// TwinCAT 3 PLC project HXR_GATT
// ProgramVersion: 3.1.4022.4
// libraries:
//   L2SI Vacuum Library, * (SLAC)
//   LCLS General, * (SLAC)
//   Tc2_ControllerToolbox, * (Beckhoff Automation GmbH)
//   Tc2_DataExchange, * (Beckhoff Automation GmbH)
//   Tc2_EtherCAT, * (Beckhoff Automation GmbH)
//   Tc2_Standard, * (Beckhoff Automation GmbH)
//   Tc2_System, * (Beckhoff Automation GmbH)
//   Tc2_Utilities, * (Beckhoff Automation GmbH)
//   Tc3_Module, * (Beckhoff Automation GmbH)
// project tree:
//   DUTs/ E_PositionState.TcDUT (not stored), ST_MPA.TcDUT, ST_PressureSensor.TcDUT
//   GVLs/ GVL_Devices.TcGVL, GVL_ILK.TcGVL, GVL_Sensors.TcGVL (not stored)
//   / PlcTask.TcTTO
//   POUs/ DIAGNOSTICS.TcPOU (not stored), FB_MPA.TcPOU, FB_PressureSensor_PX219.TcPOU (not stored), MAIN.TcPOU, PRG_ACTUATORS.TcPOU, PRG_DIFF_PUMP.TcPOU, PRG_GATT.TcPOU, PRG_GEM.TcPOU, PRG_GEM1.TcPOU, PRG_ILK.TcPOU, PRG_PMPS.TcPOU, PRG_ROOTS.TcPOU, PRG_SENSORS.TcPOU (not stored)
// real-time tasks:
//   TASK PlcTask: cycle T#10ms, priority 20, ADS port 350
// I/O:
//   DEVICE AT1L0 (EtherCAT), AmsNetId 134.79.72.124.4.1
//     PLC_AT1L0 (EK1200) [EK1200-5000 EtherCAT Power supply (2A E-Bus)]
//       PLC_EL_1 (EL2088) [EL2088 8Ch. Dig. Output 24V, 0.5A, switching to negative]
//       PLC_EL_2 (EL1088) [EL1088 8Ch. Dig. Input 24V, 3ms, negative]
//       PLC_EL_3 (EL1088) [EL1088 8Ch. Dig. Input 24V, 3ms, negative]
//       PLC_EL_4 (EL2088) [EL2088 8Ch. Dig. Output 24V, 0.5A, switching to negative]
//       PLC_EL_5 (EL1088) [EL1088 8Ch. Dig. Input 24V, 3ms, negative]
//       PLC_EL_6 (EL1088) [EL1088 8Ch. Dig. Input 24V, 3ms, negative]
//       PLC_EL_7 (EL9187) [EL9187 Potential Connection, 8 x Ground]
//       PLC_EL_8 (EL2088) [EL2088 8Ch. Dig. Output 24V, 0.5A, switching to negative]
//       PLC_EL_9 (EL1088) [EL1088 8Ch. Dig. Input 24V, 3ms, negative]
//       PLC_EL_10 (EL1088) [EL1088 8Ch. Dig. Input 24V, 3ms, negative]
//       PLC_EL_11 (EL2088) [EL2088 8Ch. Dig. Output 24V, 0.5A, switching to negative]
//       PLC_EL_12 (EL1088) [EL1088 8Ch. Dig. Input 24V, 3ms, negative]
//       PLC_EL_13 (EL1088) [EL1088 8Ch. Dig. Input 24V, 3ms, negative]
//       PLC_EL_14 (EL9187) [EL9187 Potential Connection, 8 x Ground]
//       PLC_EL_15 (EL2624) [EL2624 4Ch. Relay Output, NO (125V AC / 30V DC)]
//       PLC_EL_16 (EL2202) [EL2202 2Ch. Dig. Output 24V, 0.5A]
//       PLC_EL_17 (EL6692) [EL6692 EtherCAT Bridge terminal (Primary)]
//       PLC_EK_18 (EK1110) [EK1110 EtherCAT extension]
//     DRL_MKS (EK1100) [EK1100 EtherCAT Coupler (2A E-Bus)]
//       MKS_E1 (EL3064) [EL3064 4Ch. Ana. Input 0-10V]
//       MKS_E2 (EL3064) [EL3064 4Ch. Ana. Input 0-10V]
//       MKS_E3 (EL2794) [EL2794 4Ch. Dig. Output 24V AC/DC, 2A, short-circuit-proof]
//       MKS_E4 (EL3064) [EL3064 4Ch. Ana. Input 0-10V]
//       MKS_E5 (EL3064) [EL3064 4Ch. Ana. Input 0-10V]
//       MKS_E6 (EL2794) [EL2794 4Ch. Dig. Output 24V AC/DC, 2A, short-circuit-proof]
//       MKS_E7 (EL3064) [EL3064 4Ch. Ana. Input 0-10V]
//       MKS_E8 (EL3064) [EL3064 4Ch. Ana. Input 0-10V]
//       MKS_E9 (EL2794) [EL2794 4Ch. Dig. Output 24V AC/DC, 2A, short-circuit-proof]
//       MKS_E10 (EL3064) [EL3064 4Ch. Ana. Input 0-10V]
//       MKS_E11 (EL3064) [EL3064 4Ch. Ana. Input 0-10V]
//       MKS_E12 (EL2794) [EL2794 4Ch. Dig. Output 24V AC/DC, 2A, short-circuit-proof]
//       MKS_E13 (EL3064) [EL3064 4Ch. Ana. Input 0-10V]
//       MKS_E14 (EL3064) [EL3064 4Ch. Ana. Input 0-10V]
//       MKS_E15 (EL2794) [EL2794 4Ch. Dig. Output 24V AC/DC, 2A, short-circuit-proof]
//     L0S3_PNL_01_EB_1 (EP2338-0002) [EP2338-0002 8 Ch. Dig. Input/Output 24V, 0,5A, M12]
//     L0S3_PNL_01_EB_2 (EP2338-0002) [EP2338-0002 8 Ch. Dig. Input/Output 24V, 0,5A, M12]
//     L0S3_PNL_01_EB_3 (EP2338-0002) [EP2338-0002 8 Ch. Dig. Input/Output 24V, 0,5A, M12]
//     L0S3_PNL_01_EB_4 (EP2338-0002) [EP2338-0002 8 Ch. Dig. Input/Output 24V, 0,5A, M12]
//     L0S3_PNL_01_EB_5 (EP3174-0002) [EP3174-0002 4Ch. Ana. Input +/-10V, 0-10V, 0/4-20mA configurable]
//     L0S3_PNL_01_EB_6 (EP3174-0002) [EP3174-0002 4Ch. Ana. Input +/-10V, 0-10V, 0/4-20mA configurable]
//     L0S3_PNL_02_EB_1 (EP2338-0002) [EP2338-0002 8 Ch. Dig. Input/Output 24V, 0,5A, M12]
//     L0S3_PNL_02_EB_2 (EP2338-0002) [EP2338-0002 8 Ch. Dig. Input/Output 24V, 0,5A, M12]
//     L0S3_PNL_02_EB_3 (EP4374-0002) [EP4374-0002 2Ch. Ana. Input +/-10V, 0-10V, 0/4-20mA configurable; 2Ch. Ana. Output +/-10V, 0-10V, 0/4-20mA configurable]
//     L0S3_PNL_02_EB_4 (EP3174-0002) [EP3174-0002 4Ch. Ana. Input +/-10V, 0-10V, 0/4-20mA configurable]
//     L0S3_PNL_02_EB_5 (EP2624-0002) [EP2624-0002 4Ch. Relay Output, NO (125V AC / 30V DC)]
//     L0S3_PNL_03_EB_1 (EP2338-0002) [EP2338-0002 8 Ch. Dig. Input/Output 24V, 0,5A, M12]
//     L0S3_PNL_03_EB_2 (EP2338-0002) [EP2338-0002 8 Ch. Dig. Input/Output 24V, 0,5A, M12]
//     L0S3_PNL_03_EB_3 (EP2338-0002) [EP2338-0002 8 Ch. Dig. Input/Output 24V, 0,5A, M12]
//     L0S3_PNL_03_EB_4 (EP3174-0002) [EP3174-0002 4Ch. Ana. Input +/-10V, 0-10V, 0/4-20mA configurable]
//     L0S3_PNL_03_EB_5 (EP3174-0002) [EP3174-0002 4Ch. Ana. Input +/-10V, 0-10V, 0/4-20mA configurable]
//     L0S3_PNL_03_EB_6 (EP2624-0002) [EP2624-0002 4Ch. Relay Output, NO (125V AC / 30V DC)]
//     L0S3_PNL_03_EB_7 (EP2338-0002) [EP2338-0002 8 Ch. Dig. Input/Output 24V, 0,5A, M12]
//     L0S3_PNL_03_EB_8 (EP2624-0002) [EP2624-0002 4Ch. Relay Output, NO (125V AC / 30V DC)]
//     L0S3_PNL_03_EB_9 (EP2338-0002) [EP2338-0002 8 Ch. Dig. Input/Output 24V, 0,5A, M12]
//     L0S6_PNL_04_EB_1 (EP2338-0002) [EP2338-0002 8 Ch. Dig. Input/Output 24V, 0,5A, M12]
//     L0S6_PNL_04_EB_2 (EP3174-0002) [EP3174-0002 4Ch. Ana. Input +/-10V, 0-10V, 0/4-20mA configurable]
//     L0S6_PNL_04_EB_3 (EP4374-0002) [EP4374-0002 2Ch. Ana. Input +/-10V, 0-10V, 0/4-20mA configurable; 2Ch. Ana. Output +/-10V, 0-10V, 0/4-20mA configurable]
//     L0S6_PNL_04_EB_4 (EP2338-0002) [EP2338-0002 8 Ch. Dig. Input/Output 24V, 0,5A, M12]
//     L0S6_PNL_04_EB_5 (EP2338-0002) [EP2338-0002 8 Ch. Dig. Input/Output 24V, 0,5A, M12]
//     L0S6_PNL_04_EB_6 (EP2338-0002) [EP2338-0002 8 Ch. Dig. Input/Output 24V, 0,5A, M12]
//     L0S6_PNL_04_EB_7 (EP2338-0002) [EP2338-0002 8 Ch. Dig. Input/Output 24V, 0,5A, M12]
//     L0S6_PNL_04_EB_8 (EP2338-0002) [EP2338-0002 8 Ch. Dig. Input/Output 24V, 0,5A, M12]
//     L0S6_PNL_01_EB_1 (EP2338-0002) [EP2338-0002 8 Ch. Dig. Input/Output 24V, 0,5A, M12]
//     L0S6_PNL_01_EB_2 (EP2338-0002) [EP2338-0002 8 Ch. Dig. Input/Output 24V, 0,5A, M12]
//     L0S6_PNL_01_EB_3 (EP2338-0002) [EP2338-0002 8 Ch. Dig. Input/Output 24V, 0,5A, M12]
//     L0S6_PNL_01_EB_4 (EP3174-0002) [EP3174-0002 4Ch. Ana. Input +/-10V, 0-10V, 0/4-20mA configurable]
//     L0S6_PNL_01_EB_5 (EP3174-0002) [EP3174-0002 4Ch. Ana. Input +/-10V, 0-10V, 0/4-20mA configurable]
//     L0S6_PNL_01_EB_6 (EP2624-0002) [EP2624-0002 4Ch. Relay Output, NO (125V AC / 30V DC)]
//     L0S6_PNL_01_EB_7 (EP2338-0002) [EP2338-0002 8 Ch. Dig. Input/Output 24V, 0,5A, M12]
//     L0S6_PNL_01_EB_8 (EP2624-0002) [EP2624-0002 4Ch. Relay Output, NO (125V AC / 30V DC)]
//     L0S6_PNL_01_EB_9 (EP2338-0002) [EP2338-0002 8 Ch. Dig. Input/Output 24V, 0,5A, M12]
//     L0S6_PNL_02_EB_1 (EP2338-0002) [EP2338-0002 8 Ch. Dig. Input/Output 24V, 0,5A, M12]
//     L0S6_PNL_02_EB_2 (EP2338-0002) [EP2338-0002 8 Ch. Dig. Input/Output 24V, 0,5A, M12]
//     L0S6_PNL_02_EB_3 (EP4374-0002) [EP4374-0002 2Ch. Ana. Input +/-10V, 0-10V, 0/4-20mA configurable; 2Ch. Ana. Output +/-10V, 0-10V, 0/4-20mA configurable]
//     L0S6_PNL_02_EB_4 (EP3174-0002) [EP3174-0002 4Ch. Ana. Input +/-10V, 0-10V, 0/4-20mA configurable]
//     L0S6_PNL_02_EB_5 (EP2624-0002) [EP2624-0002 4Ch. Relay Output, NO (125V AC / 30V DC)]
//     L0S6_PNL_03_EB_1 (EP2338-0002) [EP2338-0002 8 Ch. Dig. Input/Output 24V, 0,5A, M12]
//     L0S6_PNL_03_EB_2 (EP2338-0002) [EP2338-0002 8 Ch. Dig. Input/Output 24V, 0,5A, M12]
//     L0S6_PNL_03_EB_3 (EP2338-0002) [EP2338-0002 8 Ch. Dig. Input/Output 24V, 0,5A, M12]
//     L0S6_PNL_03_EB_4 (EP2338-0002) [EP2338-0002 8 Ch. Dig. Input/Output 24V, 0,5A, M12]
//     L0S6_PNL_03_EB_5 (EP3174-0002) [EP3174-0002 4Ch. Ana. Input +/-10V, 0-10V, 0/4-20mA configurable]
//     L0S6_PNL_03_EB_6 (EP3174-0002) [EP3174-0002 4Ch. Ana. Input +/-10V, 0-10V, 0/4-20mA configurable]

CONFIGURATION HXR_GATT
    RESOURCE PLC ON TwinCAT3
        TASK PlcTask(INTERVAL := T#10ms, PRIORITY := 20);
        PROGRAM MAIN WITH PlcTask : MAIN;
    END_RESOURCE
END_CONFIGURATION

// ---- DUTs/ST_MPA.TcDUT
TYPE ST_MPA :
STRUCT
	//Readbacks
	{attribute 'pytmc' := '
    pv: INSERTED;
	io: i;
    '}
	i_bInLS	:	BOOL;
	{attribute 'pytmc' := '
    pv: RETRACTED;
	io: i;
    '}
	i_bOutLS	:	BOOL;
	//Controls
	{attribute 'pytmc' := '
    pv: INSERT_DO;
	io: i;
    '}
	q_bRetract	:	BOOL;
	{attribute 'pytmc' := '
    pv: RETRACT_DO;
	io: i;
    '}
	q_bInsert	:	BOOL;
//    q_xRetract_Do : Bool;
	
	
	//Logic and supervisory
	{attribute 'pytmc' := '
    pv: ILKOK;
	io: i;
    '}
	bILK_OK: BOOL;
	{attribute 'pytmc' := '
    pv: INSERT_OK;
	io: i;
    '}
	bInsertOK	:	BOOL;
	{attribute 'pytmc' := '
    pv: RETRACT_OK;
	io: i;
    '}
	bRetractOK	:	BOOL;
	{attribute 'pytmc' := '
    pv: INSERT_SW;
	io: io;
    '}
	bInsert_SW		:	BOOL;
	{attribute 'pytmc' := '
    pv: RETRACT_SW;
	io: io;
    '}
	bRetract_SW	:	BOOL;
	{attribute 'pytmc' := '
    pv: ERROR;
	io: io;
    '}
	bErrorPresent : BOOL;
	{attribute 'pytmc' := 
	'pv: POS_STATE ;
	type: mbbi ;
	field: ZRST RETRACTED ;
	field: ONST INSERTED ;
	field: TWST MOVING ;
	field: THST INVALID ;
	io: i
	'}
		
	eState	:	E_PositionState := INVALID;
	
END_STRUCT
END_TYPE

// ---- DUTs/ST_PressureSensor.TcDUT
TYPE ST_PressureSensor :
STRUCT
	{attribute 'pytmc' := '
    pv: PRESS;
	io: i;
    '}
	rPRESS: REAL; //This is the human-readable pressure
	{attribute 'pytmc' := '
    pv: iPRESS;
	io: i;
    '}
	iPRESS_R AT%I*: INT ; //input pressure in machine form
	{attribute 'pytmc' := '
    pv: PRESS_SP;
	io: io;
    '}	
	rPressSP: REAL ; // EPICS Pressure setpoint 
	{attribute 'pytmc' := '
    pv: MIN_SP;
	io: io;
    '}
	rMinPressSP : REAL;  // Low limit of pressure setpoint 
	{attribute 'pytmc' := '
    pv: MAX_SP;
	io: io;
    '}
	rMaxPressSP : REAL;	// High limit of pressure setpoint
	{attribute 'pytmc' := '
    pv: SCALE;
	io: io;
    '}
	rFULL_SCALE: REAL; // Full scale 
	{attribute 'pytmc' := '
    pv: ALARM;
	field: ZNAM Normal; 
	field: ONAM Alarm;
	io: i;
    '}
    xPstateAlarm : BOOL; // 0:Normal, 1:Alarm
	

END_STRUCT
END_TYPE

// ---- GVLs/GVL_Devices.TcGVL
VAR_GLOBAL
	
	(*Upstream Interface*)
	(*Gauges*)
	USG_GCC: FB_Gauge_Interface;
	DSG_GCC: FB_Gauge_Interface;
	(*Valves*)
	DSV_VGC: FB_Valve_Interface;
	
	
	(*Gauges*)
	(*EM1L0*)
	{attribute 'pytmc' :=' pv: EM1L0:GEM:GCC:10 '}
	GEM1_GCC_10 : FB_MKS422;
	{attribute 'pytmc' :=' pv: EM1L0:GEM:GPI:10 '}
	GEM1_GPI_10 : FB_MKS317;
	{attribute 'pytmc' :=' pv: EM1L0:GEM:GCC:20 '}
	GEM1_GCC_20 : FB_MKS422;
	{attribute 'pytmc' :=' pv: EM1L0:GEM:GPI:20 '}
	GEM1_GPI_20 : FB_MKS317;
	{attribute 'pytmc' :=' pv: EM1L0:GEM:GCC:30 '}
	GEM1_GCC_30 : FB_MKS422;
	{attribute 'pytmc' :=' pv: EM1L0:GEM:GPI:30 '}
	GEM1_GPI_30 : FB_MKS317;
	{attribute 'pytmc' :=' pv: EM1L0:GEM:GCC:50 '}
	GEM1_GCC_50 : FB_MKS422;
	{attribute 'pytmc' :=' pv: EM1L0:GEM:GPI:50 '}
	GEM1_GPI_50 : FB_MKS317;
	{attribute 'pytmc' :=' pv: EM1L0:GEM:GPI:11 '}
	GEM1_GPI_11 : FB_MKS275;
	{attribute 'pytmc' :=' pv: EM1L0:GEM:GPI:31 '}
	GEM1_GPI_31 : FB_MKS275;
	{attribute 'pytmc' :=' pv: EM1L0:GEM:GPI:51 '}
	GEM1_GPI_51 : FB_MKS275;
	{attribute 'pytmc' :=' pv: EM1L0:GEM:GPI:60 '}
	GEM1_GPI_60 : FB_MKS317;
	{attribute 'pytmc' :=' pv: EM1L0:GEM:GPI:61 '}
	GEM1_GPI_61 : FB_MKS275;
	{attribute 'pytmc' :=' pv: EM1L0:GEM:GPI:71 '}
	GEM1_GPI_71 : FB_MKS275;
	(*AT1L0*)
	{attribute 'pytmc' :=' pv: AT1L0:GAS:GPI:10 '}
	GATT_GPI_10 : FB_MKS317;
	(*EM2L0*)
	{attribute 'pytmc' :=' pv: EM2L0:GEM:GPI:10 '}
	GEM2_GPI_10 : FB_MKS317;
	{attribute 'pytmc' :=' pv: EM2L0:GEM:GPI:11 '}
	GEM2_GPI_11 : FB_MKS275;
	{attribute 'pytmc' :=' pv: EM2L0:GEM:GPI:21 '}
	GEM2_GPI_21 : FB_MKS275;
	{attribute 'pytmc' :=' pv: EM2L0:GEM:GCC:30 '}
	GEM2_GCC_30 : FB_MKS422;
	{attribute 'pytmc' :=' pv: EM2L0:GEM:GPI:30 '}
	GEM2_GPI_30 : FB_MKS317;
	{attribute 'pytmc' :=' pv: EM2L0:GEM:GPI:31 '}
	GEM2_GPI_31 : FB_MKS275;
	{attribute 'pytmc' :=' pv: EM2L0:GEM:GCC:50 '}
	GEM2_GCC_50 : FB_MKS422;
	{attribute 'pytmc' :=' pv: EM2L0:GEM:GPI:50 '}
	GEM2_GPI_50 : FB_MKS317;
	{attribute 'pytmc' :=' pv: EM2L0:GEM:GPI:51 '}
	GEM2_GPI_51 : FB_MKS275;
	{attribute 'pytmc' :=' pv: EM2L0:GEM:GCC:60 '}
	GEM2_GCC_60 : FB_MKS422;
	{attribute 'pytmc' :=' pv: EM2L0:GEM:GPI:60 '}
	GEM2_GPI_60 : FB_MKS317;
	{attribute 'pytmc' :=' pv: EM2L0:GEM:GPI:61 '}
	GEM2_GPI_61 : FB_MKS275;
	{attribute 'pytmc' :=' pv: EM2L0:GEM:GCC:70 '}
	GEM2_GCC_70 : FB_MKS422;
	{attribute 'pytmc' :=' pv: EM2L0:GEM:GPI:70 '}
	GEM2_GPI_70 : FB_MKS317;
	(* GAS Cell CM*)
	{attribute 'pytmc' :=' pv: AT1L0:GAS:GMP:11 '}
	GATT_GMP_11 : FB_CMR362;
	{attribute 'pytmc' :=' pv: AT1L0:GAS:GMP:10 '}
	GATT_GMP_10 : FB_GCM;
	(*GEM Gauges*)
	{attribute 'pytmc' :=' pv: EM1L0:GEM:GCM:41 '}
	GEM1_GBA_41 : FB_GCM;
	{attribute 'pytmc' :=' pv: EM1L0:GEM:GCM:42 '}
	GEM1_GBA_42 : FB_GCM;
	{attribute 'pytmc' :=' pv: EM2L0:GEM:GCM:41 '}
	GEM2_GBA_41 : FB_GCM;
	{attribute 'pytmc' :=' pv: EM2L0:GEM:GCM:42 '}
	GEM2_GBA_42 : FB_GCM;


	
	
	(*Differential Pumping section*)
	(*valves*)
	{attribute 'pytmc' :=' pv: EM1L0:GEM:VGC:10 '}
	GEM1_VGC_10: FB_VRC;
	{attribute 'pytmc' :=' pv: EM1L0:GEM:VGC:20 '}
	GEM1_VGC_20: FB_VRC;
	{attribute 'pytmc' :=' pv: EM1L0:GEM:VGC:30 '}
	GEM1_VGC_30: FB_VRC;
	{attribute 'pytmc' :=' pv: EM1L0:GEM:VGC:40 '}
	GEM1_VGC_40: FB_VRC;
	{attribute 'pytmc' :=' pv: EM1L0:GEM:VGC:50 '}
	GEM1_VGC_50: FB_VRC;
	{attribute 'pytmc' :=' pv: EM1L0:GEM:VGC:60 '}
	GEM1_VGC_60: FB_VRC;
	{attribute 'pytmc' :=' pv: EM1L0:GEM:VGC:70 '}
	GEM1_VGC_70: FB_VRC;
	{attribute 'pytmc' :=' pv: EM2L0:GEM:VGC:10 '}
	GEM2_VGC_10: FB_VRC;
	{attribute 'pytmc' :=' pv: EM2L0:GEM:VGC:20'}
	GEM2_VGC_20: FB_VRC;
	{attribute 'pytmc' :=' pv: EM2L0:GEM:VGC:30 '}
	GEM2_VGC_30: FB_VRC;
	{attribute 'pytmc' :=' pv: EM2L0:GEM:VGC:40 '}
	GEM2_VGC_40: FB_VRC;
	{attribute 'pytmc' :=' pv: EM2L0:GEM:VGC:50 '}
	GEM2_VGC_50: FB_VRC;
	{attribute 'pytmc' :=' pv: EM2L0:GEM:VGC:60 '}
	GEM2_VGC_60: FB_VRC;
	(*Turbo isolation valves*)
	{attribute 'pytmc' :=' pv: EM1L0:GAS:VRC:10 '}
	GEM1_VRC_10: FB_VRC;
	{attribute 'pytmc' :=' pv: EM1L0:GAS:VRC:20 '}
	GEM1_VRC_20: FB_VRC;
	{attribute 'pytmc' :=' pv: EM1L0:GAS:VRC:30 '}
	GEM1_VRC_30: FB_VRC;
	{attribute 'pytmc' :=' pv: EM1L0:GAS:VRC:50 '}
	GEM1_VRC_50: FB_VRC;
	{attribute 'pytmc' :=' pv: EM1L0:GAS:VRC:30 '}
	GEM2_VRC_30: FB_VRC;
	{attribute 'pytmc' :=' pv: EM1L0:GAS:VRC:50 '}
	GEM2_VRC_50: FB_VRC;
	{attribute 'pytmc' :=' pv: EM1L0:GAS:VRC:60 '}
	GEM2_VRC_60: FB_VRC;
	{attribute 'pytmc' :=' pv: EM1L0:GAS:VRC:70 '}
	GEM2_VRC_70: FB_VRC;
	(*Kashiyama Valves*)
	{attribute 'pytmc' :=' pv: EM1L0:GEM:VRC:60 '}
	GEM1_VRC_60:FB_Kashiyama_VRC;
	{attribute 'pytmc' :=' pv: EM1L0:GEM:VRC:70 '}
	GEM1_VRC_70:FB_Kashiyama_VRC;
	{attribute 'pytmc' :=' pv: EM2L0:GEM:VRC:10 '}
	GEM2_VRC_10:FB_Kashiyama_VRC;
	{attribute 'pytmc' :=' pv: EM2L0:GEM:VRC:20 '}
	GEM2_VRC_20:FB_Kashiyama_VRC;
	(*Turbo vent valves*)
	{attribute 'pytmc' :=' pv: EM1L0:GEM:VVC:20 '}
	GEM1_VVC_20: FB_TurbVentvalve_NO;
	{attribute 'pytmc' :=' pv: EM1L0:GEM:VVC:30 '}
	GEM1_VVC_30: FB_TurbVentvalve_NO;
	{attribute 'pytmc' :=' pv: EM1L0:GEM:VVC:50 '}
	GEM1_VVC_50: FB_TurbVentvalve_NO;
	{attribute 'pytmc' :=' pv: EM2L0:GEM:VVC:30 '}
	GEM2_VVC_30: FB_TurbVentvalve_NO;
	{attribute 'pytmc' :=' pv: EM2L0:GEM:VVC:50 '}
	GEM2_VVC_50: FB_TurbVentvalve_NO;
	{attribute 'pytmc' :=' pv: EM2L0:GEM:VVC:70 '}
	GEM2_VVC_70: FB_TurbVentvalve_NO;
	
	(*Gas cell vent valve*)
	{attribute 'pytmc' :=' pv: AT1L0:GAS:VVC:11 '}
	VVC_11 : FB_VVC;
	(* GAS cell needle valve*)
	{attribute 'pytmc' :=' pv: AT1L0:GAS:VCN:10 '}
	GATT_VCN_10 : FB_VCN;
	(* N2 cutt off valve *)
	{attribute 'pytmc' :=' pv: EM1L0:GEM:VVC:40'}
	GEM1_VVC_40: FB_VVC;
	{attribute 'pytmc' :=' pv: AT1L0:GAS:VVC:10 '}
	GATT_VVC_10: FB_VVC;
	{attribute 'pytmc' :=' pv: EM2L0:GEM:VVC:40 '}
	GEM2_VVC_40: FB_VVC;
	(*Pressure Control Valve*)
	{attribute 'pytmc' :=' pv: EM1L0:GEM:VPC:41 '}
	GEM1_VPC_41 : FB_MKS248;
	{attribute 'pytmc' :=' pv: EM1L0:GEM:VPC:42 '}
	GEM1_VPC_42 : FB_MKS248;
	{attribute 'pytmc' :=' pv: EM2L0:GEM:VPC:41 '}
	GEM2_VPC_41 : FB_MKS248;
	{attribute 'pytmc' :=' pv: EM2L0:GEM:VPC:42 '}
	GEM2_VPC_42 : FB_MKS248;
	
	
	
	
	{attribute 'pytmc' :=' pv: EM2L0:GEM:VGC:70 '}
	GEM2_VGC_70: FB_VGC;
	
	(*Pumps*)
	(*Turbo*)
	{attribute 'pytmc' :=' pv: EM1L0:GEM:PTM:10 '}
	GEM1_PTM_10 : FB_PTM_Agilent;
	{attribute 'pytmc' :=' pv: EM1L0:GEM:PTM:20 '}
	GEM1_PTM_20 : FB_PTM_Agilent;
	{attribute 'pytmc' :=' pv: EM1L0:GEM:PTM:30 '}
	GEM1_PTM_30 : FB_PTM_Agilent;
	{attribute 'pytmc' :=' pv: EM1L0:GEM:PTM:50 '}
	GEM1_PTM_50 : FB_PTM_Agilent;
	{attribute 'pytmc' :=' pv: EM2L0:GEM:PTM:30 '}
	GEM2_PTM_30 : FB_PTM_Agilent;
	{attribute 'pytmc' :=' pv: EM2L0:GEM:PTM:50 '}
	GEM2_PTM_50 : FB_PTM_Agilent;
	{attribute 'pytmc' :=' pv: EM2L0:GEM:PTM:60 '}
	GEM2_PTM_60 : FB_PTM_Agilent;
	{attribute 'pytmc' :=' pv: EM2L0:GEM:PTM:70 '}
	GEM2_PTM_70 : FB_PTM_Agilent;
	(*Scroll Pumps*)
	{attribute 'pytmc' :=' pv: EM1L0:GEM:PMF:20 '}
	GEM1_PMF_20 : FB_ScrollPump;
	{attribute 'pytmc' :=' pv: EM1L0:GEM:PMF:30 '}
	GEM1_PMF_30 : FB_ScrollPump;
	{attribute 'pytmc' :=' pv: EM1L0:GEM:PMF:50 '}
	GEM1_PMF_50 : FB_ScrollPump;
	{attribute 'pytmc' :=' pv: EM2L0:GEM:PMF:30 '}
	GEM2_PMF_30 : FB_ScrollPump;
	{attribute 'pytmc' :=' pv: AT1L0:GAS:PMF:50 '}
	GEM2_PMF_50 : FB_ScrollPump;
	{attribute 'pytmc' :=' pv: AT1L0:GAS:PMF:60 '}
	GEM2_PMF_60 : FB_ScrollPump;
	(*Kashyiama Dry Pumps*)
	{attribute 'pytmc' :=' pv: EM1L0:GEM:PRO:60 '}
	GEM1_PRO_60: FB_KashiyamaPump;
	{attribute 'pytmc' :=' pv: EM1L0:GEM:PRO:70 '}
	GEM1_PRO_70: FB_KashiyamaPump;
	{attribute 'pytmc' :=' pv: EM2L0:GEM:PRO:10 '}
	GEM2_PRO_10: FB_KashiyamaPump;
	{attribute 'pytmc' :=' pv: EM2L0:GEM:PRO:20 '}
	GEM2_PRO_20: FB_KashiyamaPump;
	
	
	
	
	
	(*Pneumatic actuators*)
	{attribute 'pytmc' :=' pv: AT1L0:FILTER:MPA:321 '}
	MPA_321: FB_MPA;
	{attribute 'pytmc' :=' pv: AT1L0:FILTER:MPA:322 '}
	MPA_322: FB_MPA;
	{attribute 'pytmc' :=' pv: AT1L0:FILTER:MPA:323 '}
	MPA_323: FB_MPA;
	{attribute 'pytmc' :=' pv: AT1L0:FILTER:MPA:324 '}
	MPA_324: FB_MPA;
	{attribute 'pytmc' :=' pv: AT1L0:FILTER:MPA:325 '}
	MPA_325: FB_MPA;
	{attribute 'pytmc' :=' pv: AT1L0:FILTER:MPA:326 '}
	MPA_326: FB_MPA;
	{attribute 'pytmc' :=' pv: AT1L0:FILTER:MPA:327 '}
	MPA_327: FB_MPA;
	{attribute 'pytmc' :=' pv: AT1L0:FILTER:MPA:328 '}
	MPA_328: FB_MPA;
	{attribute 'pytmc' :=' pv: AT1L0:FILTER:MPA:329 '}
	MPA_329: FB_MPA;
	
	
END_VAR

// ---- GVLs/GVL_ILK.TcGVL
VAR_GLOBAL
	

	{attribute 'pytmc' := 'pv: AT1L0:GAS:VAC:OVRDON'}
	xSystemOverrideMode	:	BOOL; (* Global system override for the GATT*)


(* Interlock related bits, local to the PLC*)
	US_Turbo_Valves_Closed:  BOOL;
	US_Turbo_Valves_Open:  BOOL;
	DS_Turbo_Valves_Closed: BOOL;
	DS_Turbo_Valves_Open:  BOOL;
	US_Turbo_Running:  BOOL;
	DS_Turbo_Running:  BOOL;
	TwinscrewPumps_Valves_Closed: BOOL;
	US_TwinscrewPumps_Valves_Open : BOOL;
	DS_TwinscrewPumps_Valves_Open : BOOL;
	US_Aperture_Closed: BOOL;
	DS_Aperture_Closed: BOOL;
	
	xUSAperturesOpnOK : BOOL;
	xDSAperturesOpnOK : BOOL;
	
	

END_VAR

// ---- POUs/MAIN.TcPOU
PROGRAM MAIN
VAR

END_VAR

(*Ethercat Diagnostics*)
DIAGNOSTICS();



(* Call all Programs*)
PRG_ILK();
PRG_DIFF_PUMP();
PRG_ROOTS();
PRG_GATT();
PRG_GEM();

END_PROGRAM

// ---- POUs/PRG_ILK.TcPOU
PROGRAM PRG_ILK
VAR
END_VAR

(*Evaluate Global Interlokcs*)

TwinscrewPumps_Valves_Closed := GEM1_VRC_60.q_stValve.i_xClsLS AND  GEM1_VRC_70.q_stValve.i_xClsLS AND GEM2_VRC_10.q_stValve.i_xClsLS AND GEM2_VRC_20.q_stValve.i_xClsLS;
US_Turbo_Valves_Closed := GEM1_VRC_10.iq_stValve.i_xClsLS AND  GEM1_VRC_20.iq_stValve.i_xClsLS AND GEM1_VRC_30.iq_stValve.i_xClsLS AND GEM1_VRC_50.iq_stValve.i_xClsLS;
DS_Turbo_Valves_Closed := GEM2_VRC_30.iq_stValve.i_xClsLS AND  GEM2_VRC_50.iq_stValve.i_xClsLS AND GEM2_VRC_60.iq_stValve.i_xClsLS AND GEM2_VRC_70.iq_stValve.i_xClsLS;
US_TwinscrewPumps_Valves_Open := (GEM1_VRC_60.q_stValve.i_xOpnLS AND GEM1_PRO_60.q_stPump.i_xIsRun) OR   (GEM1_VRC_70.q_stValve.i_xOpnLS AND GEM1_PRO_70.q_stPump.i_xIsRun);
DS_TwinscrewPumps_Valves_Open := (GEM2_VRC_10.q_stValve.i_xOpnLS AND GEM2_PRO_10.q_stPump.i_xIsRun) OR   (GEM2_VRC_20.q_stValve.i_xOpnLS AND GEM2_PRO_20.q_stPump.i_xIsRun);
US_Turbo_Valves_Open := GEM1_VRC_10.iq_stValve.i_xOpnLS AND  GEM1_VRC_20.iq_stValve.i_xOpnLS AND GEM1_VRC_30.iq_stValve.i_xOpnLS AND GEM1_VRC_50.iq_stValve.i_xOpnLS;
DS_Turbo_Valves_Open := GEM2_VRC_30.iq_stValve.i_xOpnLS AND  GEM2_VRC_50.iq_stValve.i_xOpnLS AND GEM2_VRC_60.iq_stValve.i_xOpnLS AND GEM2_VRC_70.iq_stValve.i_xOpnLS;
US_Aperture_Closed := GEM1_VGC_10.iq_stValve.i_xClsLS AND GEM1_VGC_20.iq_stValve.i_xClsLS AND GEM1_VGC_30.iq_stValve.i_xClsLS AND GEM1_VGC_40.iq_stValve.i_xClsLS AND GEM1_VGC_50.iq_stValve.i_xClsLS AND GEM1_VGC_60.iq_stValve.i_xClsLS AND GEM1_VGC_70.iq_stValve.i_xClsLS ;
DS_Aperture_Closed := GEM2_VGC_10.iq_stValve.i_xClsLS AND GEM2_VGC_20.iq_stValve.i_xClsLS AND GEM2_VGC_30.iq_stValve.i_xClsLS AND GEM2_VGC_40.iq_stValve.i_xClsLS AND GEM2_VGC_50.iq_stValve.i_xClsLS AND GEM2_VGC_60.iq_stValve.i_xClsLS; ;
US_Turbo_Running := (GEM1_PTM_10.iq_stPtm.eState = pumpRUNNING) AND (GEM1_PTM_20.iq_stPtm.eState = pumpRUNNING) AND (GEM1_PTM_30.iq_stPtm.eState = pumpRUNNING) AND (GEM1_PTM_50.iq_stPtm.eState = pumpRUNNING);
DS_Turbo_Running := (GEM2_PTM_30.iq_stPtm.eState = pumpRUNNING) AND (GEM2_PTM_50.iq_stPtm.eState = pumpRUNNING) AND (GEM2_PTM_60.iq_stPtm.eState = pumpRUNNING) AND (GEM2_PTM_70.iq_stPtm.eState = pumpRUNNING);

xUSAperturesOpnOK := NOT GEM1_VVC_40.iq_stValve.q_xOPN_DO AND NOT GATT_VVC_10.iq_stValve.q_xOPN_DO; 
xDSAperturesOpnOK := NOT GEM2_VVC_40.iq_stValve.q_xOPN_DO AND NOT GATT_VVC_10.iq_stValve.q_xOPN_DO; 

(* Link The correct override bit to the correct vacuum section*)

END_PROGRAM

// ---- POUs/PRG_DIFF_PUMP.TcPOU
PROGRAM PRG_DIFF_PUMP
VAR
END_VAR

(*Gagues*)
(*EM1L0*)
DSG_GCC(VG=>); // Downstream Gauge from Down Stream PLC System
GEM1_GPI_10(PG=>);
GEM1_GCC_10(PG:=GEM1_GPI_10.PG,IG=>);
GEM1_GPI_20(PG=>);
GEM1_GCC_20(PG:=GEM1_GPI_20.PG,IG=>);
GEM1_GPI_30(PG=>);
GEM1_GCC_30(PG:=GEM1_GPI_30.PG,IG=>);
GEM1_GPI_50(PG=>);
GEM1_GCC_50(PG:=GEM1_GPI_50.PG,IG=>);
GEM1_GPI_11(PG=>);
GEM1_GPI_31(PG=>);
GEM1_GPI_51(PG=>);
(*AT1L0*)
GEM2_GPI_30(PG=>);
GEM2_GCC_30(PG:=GEM2_GPI_30.PG,IG=>);
GEM2_GPI_31(PG=>);
GEM2_GPI_50(PG=>);
GEM2_GCC_50(PG:=GEM2_GPI_50.PG,IG=>);
GEM2_GPI_51(PG=>);
GEM2_GPI_60(PG=>);
GEM2_GCC_60(PG:=GEM2_GPI_60.PG,IG=>);
GEM2_GPI_61(PG=>);
GEM2_GPI_70(PG=>);
GEM2_GCC_70(PG:=GEM2_GPI_70.PG,IG=>);

(*VALVES*)
(*Aperture valve may open when Detector and Attenuator N2 valves are closed. Override provided *)
 (* to Include PMPS ILK with the EXTILK bit*)
(*apperture valves*)
GEM1_VGC_10(i_xExtILK_OK:=xUSAperturesOpnOK, i_xOverrideMode := xSystemOverrideMode);
GEM1_VGC_20(i_xExtILK_OK:=xUSAperturesOpnOK,i_xOverrideMode := xSystemOverrideMode);
GEM1_VGC_30(i_xExtILK_OK:=xUSAperturesOpnOK,i_xOverrideMode := xSystemOverrideMode);
GEM1_VGC_40(i_xExtILK_OK:=xUSAperturesOpnOK,i_xOverrideMode := xSystemOverrideMode);
GEM1_VGC_50(i_xExtILK_OK:=xUSAperturesOpnOK,i_xOverrideMode := xSystemOverrideMode);
GEM1_VGC_60(i_xExtILK_OK:=xUSAperturesOpnOK,i_xOverrideMode := xSystemOverrideMode);		
GEM1_VGC_70(i_xExtILK_OK:=xUSAperturesOpnOK,i_xOverrideMode := xSystemOverrideMode);
GEM2_VGC_10(i_xExtILK_OK:=xDSAperturesOpnOK,i_xOverrideMode := xSystemOverrideMode);
GEM2_VGC_20(i_xExtILK_OK:=xDSAperturesOpnOK,i_xOverrideMode := xSystemOverrideMode);
GEM2_VGC_30(i_xExtILK_OK:=xDSAperturesOpnOK,i_xOverrideMode := xSystemOverrideMode);
GEM2_VGC_40(i_xExtILK_OK:=xDSAperturesOpnOK,i_xOverrideMode := xSystemOverrideMode);	
GEM2_VGC_50(i_xExtILK_OK:=xDSAperturesOpnOK,i_xOverrideMode := xSystemOverrideMode);
GEM2_VGC_60(i_xExtILK_OK:=xDSAperturesOpnOK,i_xOverrideMode := xSystemOverrideMode);
(*downstream isolation valve*)
GEM2_VGC_70(i_stUSG := GEM2_GCC_70.IG, i_stDSG:= DSG_GCC.VG,i_xDis_DPIlk := TRUE, i_xEPS_OK := TRUE,
		i_xPMPS_OK := TRUE, i_xExt_OK := TRUE, i_xOverrideMode := xSystemOverrideMode);
DSV_VGC(VGC=>);

(*Turbo vent valves NO*)
GEM1_VVC_20(i_stPTM :=GEM1_PTM_20.iq_stPtm); 
GEM1_VVC_30(i_stPTM :=GEM1_PTM_30.iq_stPtm);
GEM1_VVC_50(i_stPTM :=GEM1_PTM_50.iq_stPtm);
GEM2_VVC_30(i_stPTM :=GEM2_PTM_30.iq_stPtm);
GEM2_VVC_50(i_stPTM :=GEM2_PTM_50.iq_stPtm);
GEM2_VVC_70(i_stPTM :=GEM2_PTM_70.iq_stPtm);


(*Turbo Isolation valves*)
 GEM1_VRC_10(i_xExtILK_OK := F_TurboGateValve_ILK(GEM1_PTM_10.iq_stPtm,GEM1_GPI_10.PG));
 GEM1_VRC_20(i_xExtILK_OK := F_TurboGateValve_ILK(GEM1_PTM_20.iq_stPtm,GEM1_GPI_20.PG));
 GEM1_VRC_30(i_xExtILK_OK := F_TurboGateValve_ILK(GEM1_PTM_30.iq_stPtm,GEM1_GPI_30.PG));
 GEM1_VRC_50(i_xExtILK_OK := F_TurboGateValve_ILK(GEM1_PTM_50.iq_stPtm,GEM1_GPI_50.PG));
 GEM2_VRC_30(i_xExtILK_OK := F_TurboGateValve_ILK(GEM2_PTM_30.iq_stPtm,GEM2_GPI_30.PG));
 GEM2_VRC_50(i_xExtILK_OK := F_TurboGateValve_ILK(GEM2_PTM_50.iq_stPtm,GEM2_GPI_50.PG));
 GEM2_VRC_60(i_xExtILK_OK := F_TurboGateValve_ILK(GEM2_PTM_60.iq_stPtm,GEM2_GPI_60.PG));
 GEM2_VRC_70(i_xExtILK_OK := F_TurboGateValve_ILK(GEM2_PTM_70.iq_stPtm,GEM2_GPI_70.PG));

(*Turbo Pumps*)
GEM1_PTM_10.i_xExtILKOk := F_TurboExtILK_NO(GEM1_PTM_10.iq_stPtm, GEM1_GPI_11.PG,
						GEM1_GPI_10.PG,GEM1_VVC_20.q_stValve,GEM1_PMF_20.iq_stPFO);
GEM1_PTM_10(i_stGauge:=GEM1_GPI_11.PG,i_rMaxBackingPressure :=0.01);
GEM1_PTM_20.i_xExtILKOk := F_TurboExtILK_NO(GEM1_PTM_20.iq_stPtm,BackingGauge:= GEM1_GPI_11.PG,
						InletGauge:=GEM1_GPI_20.PG,GEM1_VVC_20.q_stValve,GEM1_PMF_20.iq_stPFO);
GEM1_PTM_20(i_stGauge:=GEM1_GPI_11.PG,i_rMaxBackingPressure :=0.01);
GEM1_PTM_30(i_xExtILKOK:=F_TurboExtILK_NO(GEM1_PTM_30.iq_stPtm, GEM1_GPI_31.PG,
						GEM1_GPI_30.PG,GEM1_VVC_30.q_stValve,GEM1_PMF_30.iq_stPFO),
		i_stGauge:=GEM1_GPI_31.PG,i_rMaxBackingPressure :=0.01);
GEM1_PTM_50(i_xExtILKOK:=F_TurboExtILK_NO(GEM1_PTM_50.iq_stPtm, GEM1_GPI_51.PG,
						GEM1_GPI_50.PG,GEM1_VVC_50.q_stValve,GEM1_PMF_50.iq_stPFO),
		i_stGauge:=GEM1_GPI_51.PG,i_rMaxBackingPressure :=0.01);
GEM2_PTM_30(i_xExtILKOK:=F_TurboExtILK_NO(GEM2_PTM_30.iq_stPtm, GEM2_GPI_31.PG,
						GEM2_GPI_30.PG,GEM2_VVC_30.q_stValve,GEM2_PMF_30.iq_stPFO),
		i_stGauge:=GEM2_GPI_31.PG,i_rMaxBackingPressure :=0.01);
GEM2_PTM_50(i_xExtILKOK:=F_TurboExtILK_NO(GEM2_PTM_50.iq_stPtm, GEM2_GPI_51.PG,
						GEM2_GPI_50.PG,GEM2_VVC_50.q_stValve,GEM2_PMF_50.iq_stPFO),
		i_stGauge:=GEM2_GPI_51.PG,i_rMaxBackingPressure :=0.01);
GEM2_PTM_60(i_xExtILKOK:=F_TurboExtILK_NO(GEM2_PTM_60.iq_stPtm, GEM2_GPI_61.PG,
						GEM2_GPI_60.PG,GEM2_VVC_70.q_stValve,GEM2_PMF_60.iq_stPFO),
		i_stGauge:=GEM2_GPI_61.PG,i_rMaxBackingPressure :=0.01);
GEM2_PTM_70(i_xExtILKOK:=F_TurboExtILK_NO(GEM2_PTM_70.iq_stPtm, GEM2_GPI_61.PG,
						GEM2_GPI_70.PG,GEM2_VVC_70.q_stValve,GEM2_PMF_60.iq_stPFO),
		i_stGauge:=GEM2_GPI_61.PG,i_rMaxBackingPressure :=0.01);

(*Roughing pumps*)
GEM1_PMF_20(VentValve:= GEM1_VVC_20.q_stValve, TurboIsOn:= (GEM1_PTM_10.iq_stPtm.q_RunDO OR GEM1_PTM_20.iq_stPtm.q_RunDO));
GEM1_PMF_30(VentValve:= GEM1_VVC_30.q_stValve, TurboIsOn:= GEM1_PTM_30.iq_stPtm.q_RunDO);
GEM1_PMF_50(VentValve:= GEM1_VVC_50.q_stValve, TurboIsOn:= GEM1_PTM_50.iq_stPtm.q_RunDO); 
GEM2_PMF_30(VentValve:= GEM2_VVC_30.q_stValve, TurboIsOn:= GEM2_PTM_30.iq_stPtm.q_RunDO); 
GEM2_PMF_50(VentValve:= GEM2_VVC_50.q_stValve, TurboIsOn:= GEM2_PTM_50.iq_stPtm.q_RunDO); 
GEM2_PMF_60(VentValve:= GEM2_VVC_70.q_stValve, TurboIsOn:= (GEM2_PTM_60.iq_stPtm.q_RunDO OR GEM2_PTM_70.iq_stPtm.q_RunDO));

END_PROGRAM

// ---- POUs/PRG_ROOTS.TcPOU
PROGRAM PRG_ROOTS
VAR
END_VAR

(*EM1L0*)
(*Roots Pump Chamber 1*)
(*gauges*)
GEM1_GPI_60(PG=>);
GEM1_GPI_61(PG=>);
GEM1_GPI_71(PG=>);

(*Isolation Valve*)
VRC_261(Pump:=PFM_261.q_stPump,Gauge:=GEM1_GPI_60.PG,i_xExtILK_OK:=TRUE);
VRC_262(Pump:=PFM_262.q_stPump,Gauge:=GEM1_GPI_60.PG,i_xExtILK_OK:=TRUE);		


(* dry pump*)
PFM_261();
PFM_262();




(*EM2L0*)
(*Roots Pump Chamber 1*)
(*gauges*)
GEM2_GPI_10(PG=>);
GEM2_GPI_11(PG=>);
GEM2_GPI_21(PG=>);

(*Isolation Valve*)
VRC_341(Pump:=PFM_341.q_stPump,Gauge:=GEM2_GPI_10.PG,i_xExtILK_OK:=TRUE);
VRC_342(Pump:=PFM_342.q_stPump,Gauge:=GEM2_GPI_10.PG,i_xExtILK_OK:=TRUE);

(* dry pump*)
PFM_341();
PFM_342();

END_PROGRAM

// ---- POUs/PRG_GATT.TcPOU
PROGRAM PRG_GATT
VAR
	(*needle valve control position*)
	VCN_Req_Pos: REAL;
	
	fb_PID: FB_BasicPID;
	
	{attribute 'pytmc' :=' pv: AT1L0:GAS:CNTRL:SP '}
	fSetpointValue : REAL:=0.001;
	{attribute 'pytmc' :=' pv: AT1L0:GAS:CNTRL:Kp '}
	fKp : REAL:= 1.1; 
	{attribute 'pytmc' :=' pv: AT1L0:GAS:CNTRL:Tn '}
	fTn : REAL:= 0.5; 
	
	
	
	
	eMode							: E_CTRL_MODE;
	stCTRL_PID_PARAMS		: ST_CTRL_PID_PARAMS;

	eErrorId						: E_CTRL_ERRORCODES;
	bError							: BOOL;
	bARWactive					: BOOL;

	(* controller *)
	fbCTRL_PID					: FB_CTRL_PID;
	bInit							: BOOL	:= TRUE;

END_VAR

(*Gauges*)
GATT_GPI_10();
GATT_GMP_10(i_rFULL_SCALE := 2.0 (*Torr*));
GATT_GMP_11();

(*Valves*)
(*Gas Cell vent valve*)
VVC_11 (i_xExtILK_OK:= GEM2_VGC_70.iq_stValve.i_xClsLS AND DSV_VGC.VGC.i_xClsLS AND US_Turbo_Valves_Closed AND DS_Turbo_Valves_Closed AND TwinscrewPumps_Valves_Closed);

(* N2 Cutt off valve*)
GATT_VVC_10(i_xExtILK_OK := US_Aperture_Closed AND US_Turbo_Valves_Open AND US_Turbo_Running AND DS_Aperture_Closed AND DS_Turbo_Valves_Open AND US_Turbo_Running AND US_TwinscrewPumps_Valves_Open AND DS_TwinscrewPumps_Valves_Open);

(*Pressure control loop implementation*)
If(GATT_VCN_10.iq_stVCN.eValveControl = PressureControl) THEN
	//GATT_VVC_10.iq_stValve.pv_xOPN_SW := true;
	GATT_VVC_10.M_Set_OPN_SW(true);
	// check valve is open, otherwise raise error
END_IF


	
(*-------------------------------------------------------------------*)
(*        BASIC    PRG_FB_CTRL_PID               *)
(*-------------------------------------------------------------------*)
(*

fb_PID(
	fSetpointValue:= fSetpointValue, 
	fActualValue:= GATT_GBA_10.VG.rPRESS , 
	bReset:= , 
	fCtrlCycleTime:= , 
	fKp:= fKp, 
	fTn:= fTn, 
	fTv:= 0, 
	fTd:= 0, 
	fCtrlOutput=>GATT_VCN_10.i_rReqPos, 
	nErrorStatus=> );
	
*)	
(*-------------------------------------------------------------------*)
(*            PRG_FB_CTRL_PID               *)
(*-------------------------------------------------------------------*)


IF bInit
THEN
	(* init parameter struct *)
	stCTRL_PID_PARAMS.tCtrlCycleTime		:= T#10ms;
	stCTRL_PID_PARAMS.tTaskCycleTime		:= T#10ms;
	stCTRL_PID_PARAMS.fKp					:= fKp;			(* proportional gain Kp				*)
	stCTRL_PID_PARAMS.tTn					:= T#1s;		(*  Tn									*)
	stCTRL_PID_PARAMS.tTv					:= T#200ms;	(*  Tv									*)
	stCTRL_PID_PARAMS.tTd					:= T#100ms;	(*  Td									*)
	stCTRL_PID_PARAMS.fOutMaxLimit			:=  100;			(* maximum output limit				*)
	stCTRL_PID_PARAMS.fOutMinLimit			:= 0;			(* minimum output limit				*)

	(* set the mode to ACTIVE --> normal operation *)
	eMode							:= eCTRL_MODE_ACTIVE;

	(* reset the init flag *)
	bInit							:= FALSE;
END_IF

stCTRL_PID_PARAMS.fKp					:= fKp;			
stCTRL_PID_PARAMS.tTn					:= T#1s;	

(* call controller *)
fbCTRL_PID(		fSetpointValue		:= fSetpointValue,
					fActualValue		:= GATT_GMP_10.VG.rPRESS, // Pressure gauge selection
					fManSyncValue	:= ,
					bSync				:= ,
					eMode				:= eMode,
					bHold				:= ,
					stParams			:= stCTRL_PID_PARAMS,
					fOut				=> (VCN_Req_Pos),
					bARWactive		=> bARWactive,
					eErrorId			=> eErrorId,
					bError				=> bError
				);


(*flow control valve*)
GATT_VCN_10(i_xExtIlkOK:= TRUE,i_ReqPos:= VCN_Req_Pos);

END_PROGRAM

// ---- POUs/PRG_GEM.TcPOU
PROGRAM PRG_GEM
VAR
	
	(*Pressure Control valve  position*)
	VPC_241_Req_Pos: REAL;
	VPC_242_Req_Pos: REAL;
	
	VPC_361_Req_Pos: REAL;
	VPC_362_Req_Pos: REAL;
	
END_VAR

(* GEM 1*)

(*Gauges*)
GEM1_GBA_41(i_rFULL_SCALE := 10.0 (*Torr*));
GEM1_GBA_42(i_rFULL_SCALE := 0.05 (*Torr*));

(* N2 Cut Off Valves *)
GEM1_VVC_40(i_xExtILK_OK:= US_Aperture_Closed AND US_Turbo_Valves_Open AND US_Turbo_Running); 

(*Flow Control Valves*)
GEM1_VPC_41 (i_xExtIlkOK := TRUE, i_rReqPos:= VPC_241_Req_Pos);
GEM1_VPC_42 (i_xExtIlkOK := TRUE, i_rReqPos:= VPC_242_Req_Pos);


(* GEM 2*)

(*Gauges*)
GEM2_GBA_41(i_rFULL_SCALE := 2.0 (*Torr*));
GEM2_GBA_42(i_rFULL_SCALE := 0.05 (*Torr*));
(* N2 Cut Off Valves *)
GEM2_VVC_40(i_xExtILK_OK:= DS_Aperture_Closed AND DS_Turbo_Valves_Open AND DS_Turbo_Running); 


(*Flow Control Valves*)
GEM2_VPC_41(i_xExtIlkOK := TRUE, i_rReqPos:= VPC_361_Req_Pos);
GEM2_VPC_42(i_xExtIlkOK := TRUE, i_rReqPos:= VPC_362_Req_Pos);

(*Control Loop to be implemented*)

END_PROGRAM

// ---- POUs/FB_MPA.TcPOU
FUNCTION_BLOCK FB_MPA
VAR_INPUT
	(*EPS Interlock Bits*)
	ibInsertOK: BOOL;
	ibRetractOK: BOOL;
	ibPMPS_OK:BOOL;
	ibOverrideInterlock:BOOL; (*if true interlocks are ignored*)
END_VAR
VAR_OUTPUT
	{attribute 'pytmc' := '
    pv:
	'}
	q_stAct 	:	ST_MPA;
	{attribute 'pytmc' := '
    pv: MPS_FAULT
	'}
	xMPS_OK:BOOL;
	{attribute 'pytmc' := '
    pv: MOT_DONE
	'}
	xDone:Bool; // Motion is Done 
END_VAR

VAR
	
	(*Init*)
	xFirstPass	:	BOOL;
	fbFSInit		:	R_TRIG;
	
	(* Timeouts*)
	tTimeOutDuration: TIME:= T#5S;
	tInserttimeout: TON;
	tRetracttimeout:TON;
	
	(*IO*)
	i_xInsertedLS	AT%I*: BOOL;
	i_xRetractedLS	AT%I*: BOOL;
	q_xInsert_DO	AT%Q*: BOOL;
	q_xRetract_DO	AT%Q*: BOOL;
	
END_VAR


(*Initialize*)
fbFSInit( CLK := TRUE, Q => xFirstPass);
(*IO Mapping*)
ACT_IO();

IF xFirstPass THEN
	q_stAct.eState := INVALID;
	q_stAct.bRetract_SW := FALSE;
	q_stAct.bInsert_SW := FALSE;
END_IF


(* Manage States*)
IF q_stAct.i_bInLS AND  q_stAct.i_bOutLS THEN
	q_stAct.eState:=INVALID;
ELSIF NOT q_stAct.i_bInLS AND q_stAct.i_bOutLS AND q_stAct.q_bRetract THEN 
	q_stAct.eState:=RETRACTED;
ELSIF q_stAct.i_bInLS AND NOT q_stAct.i_bOutLS AND q_stAct.q_bInsert THEN 
	q_stAct.eState:=INSERTED;
ELSIF NOT q_stAct.i_bInLS AND NOT q_stAct.i_bOutLS THEN 
	q_stAct.eState:=MOVING;
ELSE
	q_stAct.eState:=INVALID;
END_IF

(*Set the Done signal*)
xDone := (q_stAct.bRetract_SW AND q_stAct.eState=RETRACTED) OR (q_stAct.eState=INSERTED AND q_stAct.bInsert_SW);
	

(*MPS FAULT*)
//xMPS_OK := (q_stAct.eState=INSERTED);

(*PMPS PERMISSION*)

(*Actuate the device*)
q_stAct.q_bRetract := q_stAct.bRetractOK AND q_stAct.bRetract_SW;
q_stAct.q_bInsert := q_stAct.bInsertOK AND q_stAct.bInsert_SW;

IF q_stAct.q_bInsert THEN
	q_stAct.q_bRetract := FALSE;
	q_stAct.bRetract_SW:= FALSE;
ELSIF q_stAct.q_bRetract THEN
	q_stAct.q_bInsert := FALSE;
	q_stAct.bInsert_SW:= FALSE;
END_IF;


(*Timers*)
tInserttimeout(IN:= q_stAct.q_bInsert, PT := tTimeOutDuration );
tRetracttimeout(IN:= q_stAct.q_bRetract, PT := tTimeOutDuration);

///Check moving postion timout
IF NOT q_stAct.i_bInLS AND tInserttimeout.Q THEN 
	q_stAct.bErrorPresent := TRUE;
ELSIF NOT q_stAct.i_bOutLS AND tRetracttimeout.Q THEN 
	q_stAct.bErrorPresent := TRUE; 
END_IF


(*Soft IO Mapping*)
ACT_IO();

ACTION ACT_IO:
(*Inputs*)
q_stAct.i_bInLS :=  i_xInsertedLS;
q_stAct.i_bOutLS := i_xRetractedLS;
	
(*outputs*)
q_xInsert_DO:=q_stAct.q_bInsert;
q_xRetract_DO:=q_stAct.q_bRetract;
END_ACTION

END_FUNCTION_BLOCK

// ---- POUs/PRG_ACTUATORS.TcPOU
PROGRAM PRG_ACTUATORS
VAR
END_VAR

MPA_321();
MPA_322();
MPA_323();
MPA_324();
MPA_325();
MPA_326();
MPA_327();
MPA_328();
MPA_329();

END_PROGRAM

// ---- POUs/PRG_GEM1.TcPOU
FUNCTION_BLOCK PRG_GEM1
VAR_INPUT
END_VAR
VAR_OUTPUT
END_VAR
VAR
END_VAR

END_FUNCTION_BLOCK

// ---- POUs/PRG_PMPS.TcPOU
PROGRAM PRG_PMPS
VAR
END_VAR

END_PROGRAM
